% RSLogix 500 project P8_BAK009.RSS, saved by version 8.10.00.18 %
PROJECT "UNTITLED"    % processor: Bul.1763 MicroLogix 1100 Series B %

PROGRAM FILES
  LAD 2   4 rungs
  LAD 3 "IO'S"  3 rungs
  LAD 4 "CTRL"  11 rungs

DATA FILES
  O0 OUTPUT  4 elements
  I1 INPUT  6 elements
  S2 STATUS  66 elements
  B3 BINARY  1 elements
  T4 TIMER  1 elements
  C5 COUNTER  1 elements
  R6 CONTROL  1 elements
  N7 INTEGER  8 elements
  F8 FLOAT  2 elements

LADDER 2
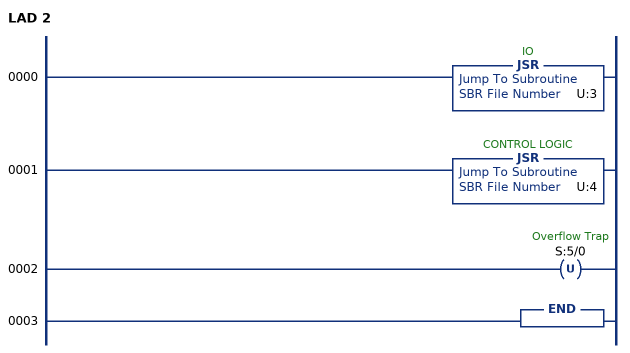
% Rung: 0 %
SOR JSR U:3 EOR
%   U:3  "IO" %
% Rung: 1 %
SOR JSR U:4 EOR
%   U:4  "CONTROL LOGIC" %
% Rung: 2 %
SOR OTU S:5/0 EOR
%   S:5/0  "Overflow Trap" %
% Rung: 3 %
SOR END EOR

LADDER 3 "IO'S"
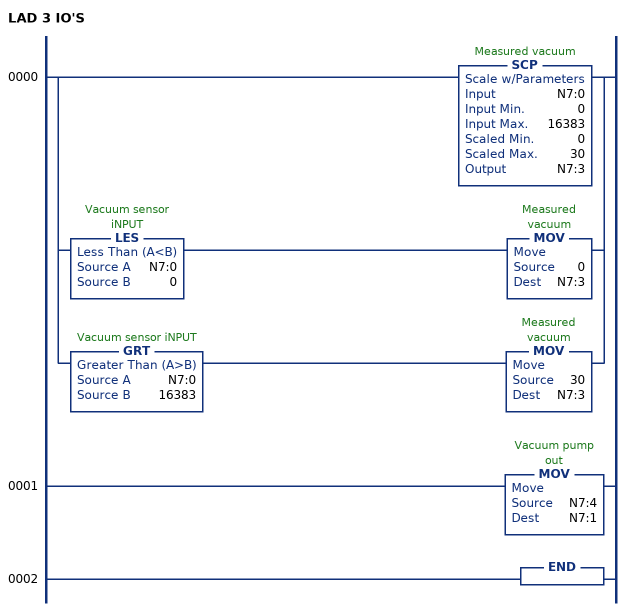
% Rung: 0 %
SOR BST SCP N7:0 0 16383 0 30 N7:3 NXB LES N7:0 0 MOV 0 N7:3 NXB GRT N7:0 16383 MOV 30 N7:3 BND EOR
%   N7:0  "Vacuum sensor iNPUT" %
%   N7:3  "Measured vacuum" %
% Rung: 1 %
SOR MOV N7:4 N7:1 EOR
%   N7:4  "CALCULATED PUMP SPEEED" %
%   N7:1  "Vacuum pump out" %
% Rung: 2 %
SOR END EOR

LADDER 4 "CTRL"
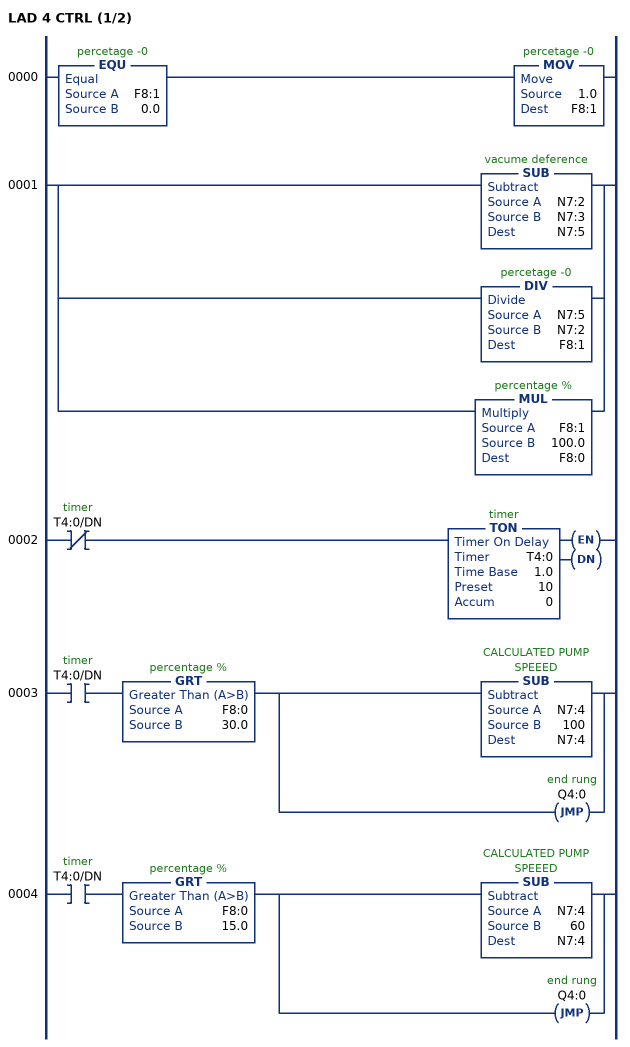
% Rung: 0 %
SOR EQU F8:1 0.0 MOV 1.0 F8:1 EOR
%   F8:1  "percetage -0" %
% Rung: 1 %
SOR BST SUB N7:2 N7:3 N7:5 NXB DIV N7:5 N7:2 F8:1 NXB MUL F8:1 100.0 F8:0 BND EOR
%   N7:2  "Vacuum setpoint" %
%   N7:3  "Measured vacuum" %
%   N7:5  "vacume deference" %
%   F8:1  "percetage -0" %
%   F8:0  "percentage %" %
% Rung: 2 %
SOR XIO T4:0/DN TON T4:0 1.0 10 0 EOR
%   T4:0  "timer" %
% Rung: 3 %
SOR XIC T4:0/DN GRT F8:0 30.0 BST SUB N7:4 100 N7:4 NXB JMP Q4:0 BND EOR
%   T4:0  "timer" %
%   F8:0  "percentage %" %
%   N7:4  "CALCULATED PUMP SPEEED" %
%   Q4:0  "end rung" %
% Rung: 4 %
SOR XIC T4:0/DN GRT F8:0 15.0 BST SUB N7:4 60 N7:4 NXB JMP Q4:0 BND EOR
%   T4:0  "timer" %
%   F8:0  "percentage %" %
%   N7:4  "CALCULATED PUMP SPEEED" %
%   Q4:0  "end rung" %

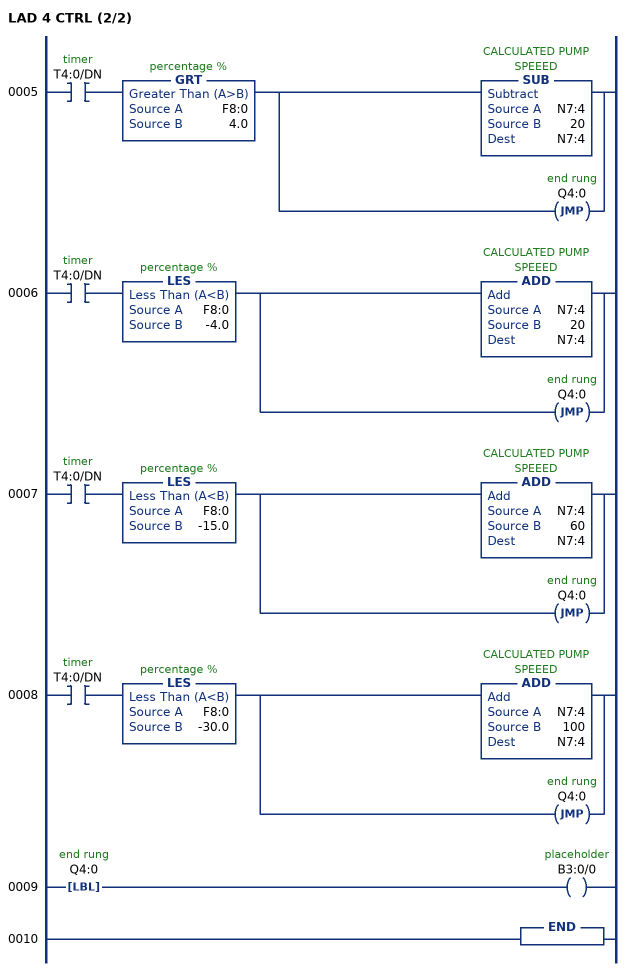
% Rung: 5 %
SOR XIC T4:0/DN GRT F8:0 4.0 BST SUB N7:4 20 N7:4 NXB JMP Q4:0 BND EOR
%   T4:0  "timer" %
%   F8:0  "percentage %" %
%   N7:4  "CALCULATED PUMP SPEEED" %
%   Q4:0  "end rung" %
% Rung: 6 %
SOR XIC T4:0/DN LES F8:0 -4.0 BST ADD N7:4 20 N7:4 NXB JMP Q4:0 BND EOR
%   T4:0  "timer" %
%   F8:0  "percentage %" %
%   N7:4  "CALCULATED PUMP SPEEED" %
%   Q4:0  "end rung" %
% Rung: 7 %
SOR XIC T4:0/DN LES F8:0 -15.0 BST ADD N7:4 60 N7:4 NXB JMP Q4:0 BND EOR
%   T4:0  "timer" %
%   F8:0  "percentage %" %
%   N7:4  "CALCULATED PUMP SPEEED" %
%   Q4:0  "end rung" %
% Rung: 8 %
SOR XIC T4:0/DN LES F8:0 -30.0 BST ADD N7:4 100 N7:4 NXB JMP Q4:0 BND EOR
%   T4:0  "timer" %
%   F8:0  "percentage %" %
%   N7:4  "CALCULATED PUMP SPEEED" %
%   Q4:0  "end rung" %
% Rung: 9 %
SOR LBL Q4:0 OTE B3:0/0 EOR
%   Q4:0  "end rung" %
%   B3:0/0  "placeholder" %
% Rung: 10 %
SOR END EOR

OTHER DOCUMENTED ADDRESSES
  N7:6  "Pre-percentage"
  N7:7  "percentage"

DATA TABLE (non-zero values as saved)
DATA T4
% .PRE .ACC %
% T4:0 % 10 0
DATA F8
% F8:0 % 0 1
